FUNCTION_BLOCK SensorReader
VAR_INPUT
	mxEnable: BOOL;
END_VAR
VAR_OUTPUT
	Product:STRING;
END_VAR
VAR
	SensorReader:BYTE;
END_VAR

IF mxEnable THEN
	SensorReader.1:=gvl.ixInductiveSensor1;
	SensorReader.2:=gvl.ixInductiveSensor2;
	SensorReader.3:=gvl.ixInductiveSensor3;
	SensorReader.4:=gvl.ixInductiveSensor4;
END_IF

IF SensorReader = 0 OR SensorReader = 4 OR SensorReader = 2 OR SensorReader = 6 THEN
 	Product:='InvalidPart';
END_IF

IF SensorReader=16 THEN
	Product:='Blue Container';
END_IF

IF SensorReader=8 THEN
	Product:='Yellow Container';
END_IF

IF SensorReader=24 THEN
	Product:='Red Container';
END_IF

IF SensorReader=20 THEN
	Product:='Blue Cylinder';
END_IF

IF SensorReader=12 THEN
	Product:='Blue Octagon';
END_IF

IF SensorReader=28 THEN
	Product:='Blue Plate';
END_IF

IF SensorReader=18 THEN
	Product:='Yellow Cylinder';
END_IF

IF SensorReader=10 THEN
	Product:='Yellow Octagon';
END_IF

IF SensorReader=26 THEN
	Product:='Yellow Plate';
END_IF

IF SensorReader=22 THEN
	Product:='Red Cylinder';
END_IF

IF SensorReader=14 THEN
	Product:='Red Octagon';
END_IF

IF SensorReader=30 THEN
	Product:='Red Plate';
END_IF

END_FUNCTION_BLOCK

(* stored: Version 1.1.0.1, ProductVersion 3.1.4024.12
   POU SensorReader: Id {aa91b23e-85b8-4465-b57d-fffd9118ff41}, SpecialFunc None *)
